{attribute 'linkalways'} 
{attribute 'no_explicit_call' := 'This FB is a CLASS and must be accessed using methods or properties'}
{attribute 'enable_dynamic_creation'}
FUNCTION_BLOCK Node_F_VN_RegionsMSER EXTENDS VisionNode
VAR
    ipSrcImage : _ITcVnImage;
    ipRegions : _ITcVnContainer;
    ipBoundingBoxes : _ITcVnContainer;
    hrPrev : _HRESULT(S_OK);
	hresult : _HRESULT(S_OK);
END_VAR

METHOD PUBLIC  Clone : I_Node
VAR
	pNode : POINTER TO Node_F_VN_RegionsMSER;
END_VAR
pNode := __NEW(Node_F_VN_RegionsMSER);
Clone := pNode^;
END_METHOD

METHOD FB_init : BOOL
VAR_INPUT
	bInitRetains : BOOL; // if TRUE, the retain variables are initialized (warm start / cold start)
	bInCopyCode : BOOL;  // if TRUE, the instance afterwards gets moved into the copy code (online change)
END_VAR
AddInput('ipSrcImage', ipSrcImage);
AddInput('hrPrev', hrPrev);
AddOutput('ipRegions', ipRegions);
AddOutput('ipBoundingBoxes', ipBoundingBoxes);
AddOutput('hresult',hresult);
END_METHOD

METHOD PROTECTED OnExecute : HRESULT
hresult.Value := F_VN_RegionsMSER(
	ipSrcImage := ipSrcImage.Value,
    ipRegions := ipRegions.Value,
    ipBoundingBoxes := ipBoundingBoxes.Value,
	hrPrev:= hrPrev.Value);
END_METHOD

METHOD PUBLIC PreExecutionCheck
VAR_INPUT
	Check : I_PreExecutionChecks;
END_VAR
Check.IsTrue(ipSrcImage.IsValid, 'ipSrcImage must contain an image');
END_METHOD

END_FUNCTION_BLOCK

(* stored: Version 1.1.0.1, ProductVersion 3.1.4024.13
   POU Node_F_VN_RegionsMSER: Id {b097f75e-0646-40d5-b3da-c32654254f2c}, SpecialFunc None
   Folder Constructor: Id {8c9e1bcc-cc66-4e1c-9ef4-f1d5a2fcab01}
   Method Clone: Id {cd81450b-28c2-41ab-b388-1b4b3e5bee38}
   Method FB_init: Id {48a59821-05a4-4e0b-a8ab-70d86088ce84}
   Method OnExecute: Id {5c28876d-827b-4b82-b0a6-a76aa2e6ad69}
   Method PreExecutionCheck: Id {90d9de13-65a5-44cf-8476-3daeeb8c3770} *)
